// TIA Portal V20 export
FUNCTION_BLOCK "05 T10 LANT Sequence"   // FB1593, GRAPH
// stored: AutoNumber false, GraphVersion 6.0, InitialValuesAcquisition false, SetENOAutomatically false
   // inherited from GRAPH_BASE
   VAR_INPUT
      OFF_SQ : Bool := false;
      INIT_SQ : Bool := false;
      ACK_EF : Bool := false;
      S_PREV : Bool := false;
      S_NEXT : Bool := false;
      SW_AUTO : Bool := false;
      SW_TAP : Bool := false;
      SW_TOP : Bool := false;
      SW_MAN : Bool := false;
      S_SEL : Int := 0;
      S_ON : Bool := false;
      S_OFF : Bool := false;
      T_PUSH : Bool := false;
   END_VAR
   VAR_OUTPUT
      S_NO : Int := 0;
      S_MORE : Bool := false;
      S_ACTIVE : Bool := false;
      ERR_FLT : Bool := false;
      AUTO_ON : Bool := false;
      TAP_ON : Bool := false;
      TOP_ON : Bool := false;
      MAN_ON : Bool := false;
   END_VAR
BEGIN
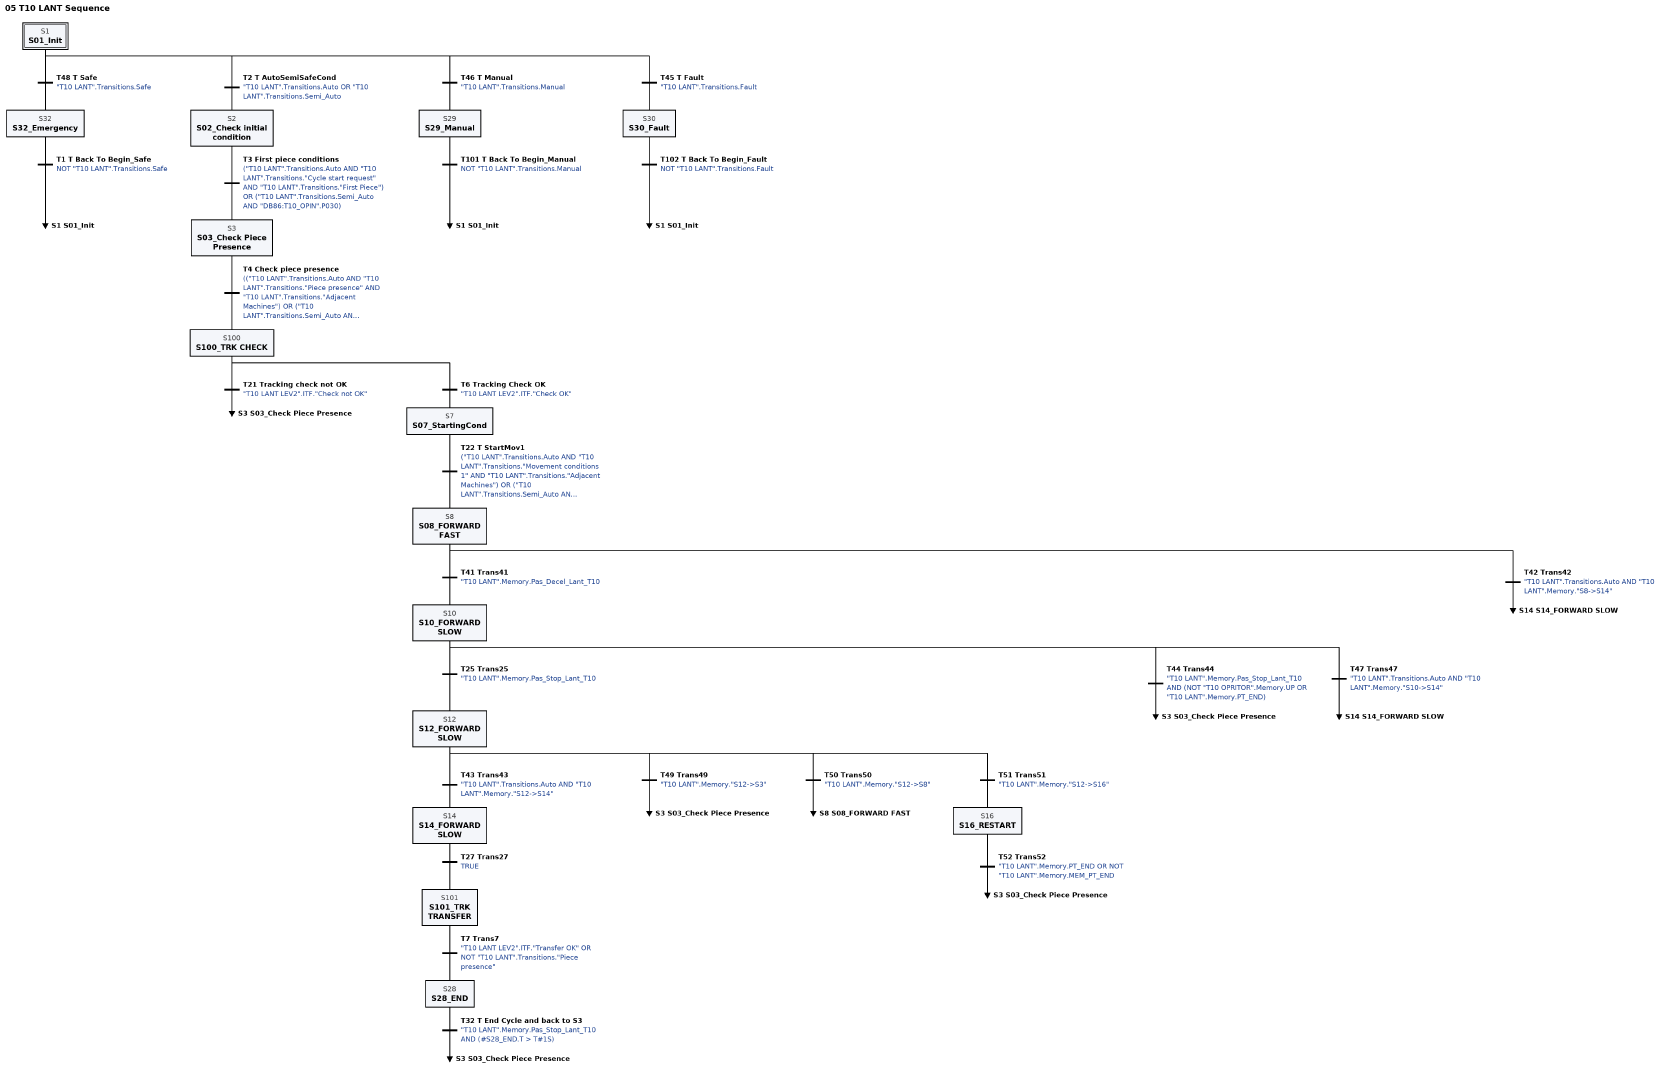
   // permanent pre-instructions
   NETWORK 1
      "01 T10 LANT Alarms"();
   NETWORK 2
      "02 T10 LANT HMI"();
   NETWORK 3
      "03 T10 LANT Aux"();
   NETWORK 4
      "04 T10 LANT Transitions"();

   // sequencer 1
   INITIAL_STEP S01_Init:   // S1, max time T#10S, warning time T#7S
   END_STEP
   TRANSITION "T Safe" FROM S01_Init TO S32_Emergency   // T48
      := "T10 LANT".Transitions.Safe;
   END_TRANSITION
   TRANSITION "T AutoSemiSafeCond" FROM S01_Init TO "S02_Check initial condition"   // T2
      := "T10 LANT".Transitions.Auto OR "T10 LANT".Transitions.Semi_Auto;
   END_TRANSITION
   TRANSITION "T Manual" FROM S01_Init TO S29_Manual   // T46
      := "T10 LANT".Transitions.Manual;
   END_TRANSITION
   TRANSITION "T Fault" FROM S01_Init TO S30_Fault   // T45
      := "T10 LANT".Transitions.Fault;
   END_TRANSITION
   STEP "S03_Check Piece Presence":   // S3, max time T#10S, warning time T#7S
   END_STEP
   TRANSITION "Check piece presence" FROM "S03_Check Piece Presence" TO "S100_TRK CHECK"   // T4
      := (("T10 LANT".Transitions.Auto AND "T10 LANT".Transitions."Piece presence" AND "T10 LANT".Transitions."Adjacent Machines") OR ("T10 LANT".Transitions.Semi_Auto AND "DB86:T10_OPIN".P030)) AND (("DA SOSTITUIRE STEVEN"."FK Ready" AND "DA SOSTITUIRE STEVEN"."KASTO 1 I/O E359.1") OR NOT "T10 LANT".Memory.PT_END) AND NOT "T10 LANT".Transitions.Pause;
   END_TRANSITION
   STEP S32_Emergency:   // S32, max time T#10S, warning time T#7S
   END_STEP
   TRANSITION "T Back To Begin_Safe" FROM S32_Emergency TO S01_Init   // T1, jump
      := NOT "T10 LANT".Transitions.Safe;
   END_TRANSITION
   STEP S29_Manual:   // S29, max time T#10S, warning time T#7S
   END_STEP
   TRANSITION "T Back To Begin_Manual" FROM S29_Manual TO S01_Init   // T101, jump
      := NOT "T10 LANT".Transitions.Manual;
   END_TRANSITION
   STEP "S02_Check initial condition":   // S2, max time T#10S, warning time T#7S
   END_STEP
   TRANSITION "First piece conditions" FROM "S02_Check initial condition" TO "S03_Check Piece Presence"   // T3
      := ("T10 LANT".Transitions.Auto AND "T10 LANT".Transitions."Cycle start request" AND "T10 LANT".Transitions."First Piece") OR ("T10 LANT".Transitions.Semi_Auto AND "DB86:T10_OPIN".P030);
   END_TRANSITION
   STEP S30_Fault:   // S30, max time T#10S, warning time T#7S
   END_STEP
   TRANSITION "T Back To Begin_Fault" FROM S30_Fault TO S01_Init   // T102, jump
      := NOT "T10 LANT".Transitions.Fault;
   END_TRANSITION
   STEP S28_END:   // S28, max time T#10S, warning time T#7S
   END_STEP
   TRANSITION "T End Cycle and back to S3" FROM S28_END TO "S03_Check Piece Presence"   // T32, jump: Assenza pezzo o ok da robot
      := "T10 LANT".Memory.Pas_Stop_Lant_T10 AND (#S28_END.T > T#1S);
   END_TRANSITION
   STEP "S10_FORWARD SLOW":   // S10, max time T#10S, warning time T#7S
   END_STEP
   TRANSITION Trans25 FROM "S10_FORWARD SLOW" TO "S12_FORWARD SLOW"   // T25
      := "T10 LANT".Memory.Pas_Stop_Lant_T10;
   END_TRANSITION
   TRANSITION Trans44 FROM "S10_FORWARD SLOW" TO "S03_Check Piece Presence"   // T44, jump
      := "T10 LANT".Memory.Pas_Stop_Lant_T10 AND (NOT "T10 OPRITOR".Memory.UP OR "T10 LANT".Memory.PT_END);
   END_TRANSITION
   TRANSITION Trans47 FROM "S10_FORWARD SLOW" TO "S14_FORWARD SLOW"   // T47, jump
      := "T10 LANT".Transitions.Auto AND "T10 LANT".Memory."S10->S14";
   END_TRANSITION
   STEP "S14_FORWARD SLOW":   // S14, max time T#10S, warning time T#7S
   END_STEP
   TRANSITION Trans27 FROM "S14_FORWARD SLOW" TO "S101_TRK TRANSFER"   // T27
      := TRUE;
   END_TRANSITION
   STEP "S100_TRK CHECK":   // S100, max time T#10S, warning time T#7S
   END_STEP
   TRANSITION "Tracking check not OK" FROM "S100_TRK CHECK" TO "S03_Check Piece Presence"   // T21, jump
      := "T10 LANT LEV2".ITF."Check not OK";
   END_TRANSITION
   TRANSITION "Tracking Check OK" FROM "S100_TRK CHECK" TO S07_StartingCond   // T6
      := "T10 LANT LEV2".ITF."Check OK";
   END_TRANSITION
   STEP "S101_TRK TRANSFER":   // S101, max time T#10S, warning time T#7S
   END_STEP
   TRANSITION Trans7 FROM "S101_TRK TRANSFER" TO S28_END   // T7
      := "T10 LANT LEV2".ITF."Transfer OK" OR NOT "T10 LANT".Transitions."Piece presence";
   END_TRANSITION
   STEP S07_StartingCond:   // S7, max time T#10S, warning time T#7S
   END_STEP
   TRANSITION "T StartMov1" FROM S07_StartingCond TO "S08_FORWARD FAST"   // T22
      := ("T10 LANT".Transitions.Auto AND "T10 LANT".Transitions."Movement conditions 1" AND "T10 LANT".Transitions."Adjacent Machines") OR ("T10 LANT".Transitions.Semi_Auto AND "DB86:T10_OPIN".P030);
   END_TRANSITION
   STEP S16_RESTART:   // S16, max time T#10S, warning time T#7S
   END_STEP
   TRANSITION Trans52 FROM S16_RESTART TO "S03_Check Piece Presence"   // T52, jump
      := "T10 LANT".Memory.PT_END OR NOT "T10 LANT".Memory.MEM_PT_END;
   END_TRANSITION
   STEP "S08_FORWARD FAST":   // S8, max time T#10S, warning time T#7S
   END_STEP
   TRANSITION Trans41 FROM "S08_FORWARD FAST" TO "S10_FORWARD SLOW"   // T41
      := "T10 LANT".Memory.Pas_Decel_Lant_T10;
   END_TRANSITION
   TRANSITION Trans42 FROM "S08_FORWARD FAST" TO "S14_FORWARD SLOW"   // T42, jump
      := "T10 LANT".Transitions.Auto AND "T10 LANT".Memory."S8->S14";
   END_TRANSITION
   STEP "S12_FORWARD SLOW":   // S12, max time T#10S, warning time T#7S
   END_STEP
   TRANSITION Trans43 FROM "S12_FORWARD SLOW" TO "S14_FORWARD SLOW"   // T43
      := "T10 LANT".Transitions.Auto AND "T10 LANT".Memory."S12->S14";
   END_TRANSITION
   TRANSITION Trans49 FROM "S12_FORWARD SLOW" TO "S03_Check Piece Presence"   // T49, jump
      := "T10 LANT".Memory."S12->S3";
   END_TRANSITION
   TRANSITION Trans50 FROM "S12_FORWARD SLOW" TO "S08_FORWARD FAST"   // T50, jump
      := "T10 LANT".Memory."S12->S8";
   END_TRANSITION
   TRANSITION Trans51 FROM "S12_FORWARD SLOW" TO S16_RESTART   // T51
      := "T10 LANT".Memory."S12->S16";
   END_TRANSITION

   // permanent post-instructions
   NETWORK 1
      "06 T10 LANT Output"();
   NETWORK 2
      "07 T10 LANT LEV2"();
END_FUNCTION_BLOCK
